FUNCTION_BLOCK FB_Inverter IMPLEMENTS I_Inverter
VAR_INPUT
	UnitID		: BYTE;	
	id			: UINT;
END_VAR
VAR_OUTPUT
END_VAR
VAR
	TargetSpeed			: REAL;
	fActualSpeed AT %I*	: REAL;
	bBrake 		 AT %Q* : BOOL;
	bVFD		 AT %Q* : BOOL;
	bReverse	 AT %Q* : BOOL;
	bReset		 AT %Q*	: BOOL;
	nErrId				: INT;
	
	fbInterfaceMbus		: FB_Interface_MbRtu;
	bExecute 			: BOOL;
	bStop				: BOOL;
	WriteVal1			: REAL;
	WriteVal2			: REAL;
	WriteVal3			: REAL;
END_VAR

fbInterfaceMbus(
	UnitID:= UnitID, 
	bExecute:= bExecute, 
	bStop:= bStop, 
	bReset:= bReset,
	idDevice := id,
	fTargetSpeed:= fTargetSpeed);

PROPERTY ActualSpeed : REAL
GET
ActualSpeed := fActualSpeed/100;
END_GET
END_PROPERTY

PROPERTY bIsMove : BOOL
GET
IF bVFD OR bReverse THEN 
	bIsMove := TRUE;
ELSIF NOT bVFD AND NOT bReverse THEN
	bIsMove := FALSE;
END_IF
END_GET
END_PROPERTY

PROPERTY fTargetSpeed : REAL
GET
fTargetSpeed := TargetSpeed;
END_GET
SET
TargetSpeed := fTargetSpeed;
END_SET
END_PROPERTY

METHOD Reset : BOOL
VAR_INPUT
END_VAR
bStop	 := FALSE;
bReset	 := TRUE;
bExecute := FALSE;
bVFD	 := FALSE;
END_METHOD

METHOD Reverse : BOOL
VAR_INPUT
END_VAR
bExecute := TRUE;
bStop	 := FALSE;
bReset	 := FALSE;
bReverse := TRUE;
bVFD 	 := false;
END_METHOD

METHOD Start : BOOL
VAR_INPUT
END_VAR
bExecute := TRUE;
bStop	 := FALSE;
bReset	 := FALSE;
bVFD	 := TRUE;
bReverse := false;
END_METHOD

METHOD Stop : BOOL
VAR_INPUT
END_VAR
bExecute := FALSE;
bStop	 := TRUE;
bReset	 := FALSE;
bVFD	 := FALSE;
bReverse := false;
END_METHOD

END_FUNCTION_BLOCK

(* stored: Version 1.1.0.1, ProductVersion 3.1.4024.12
   POU FB_Inverter: Id {fac70b65-6562-4a81-8070-9a789707e623}, SpecialFunc None
   Property ActualSpeed: Id {d2a175f0-8795-465e-b91c-9e487d4b40fa}
   Get Get: Id {61386726-836d-440b-b616-356d5f2fe22a}
   Property bIsMove: Id {75908c6f-195f-415f-a3e4-8a7137821b78}
   Get Get: Id {47cab446-da80-44b8-8b5c-8ab325dd5968}
   Property fTargetSpeed: Id {dd0d149b-b085-424d-953b-b801f80fb27a}
   Get Get: Id {a4e514c8-4b39-4312-94ff-fba384ab652d}
   Set Set: Id {54af87fd-3a9b-46a4-9b97-c87bfef50503}
   Method Reset: Id {28b24c92-a680-49d6-8321-f68524566246}
   Method Reverse: Id {d22f891c-feb4-4e6b-a9f7-77e2a23e318c}
   Method Start: Id {5753aa38-0732-4c48-8288-db7180a0f573}
   Method Stop: Id {21eba6b6-6a34-47fc-8935-a20df8f47973} *)
